PROGRAM AxisDriver
VAR
    fbReset : MC_Reset;  // PLCopen reset
    fbPower : MC_Power;  // PLCopen enable power
    bEnable : BOOL := TRUE;
END_VAR

// Reset faults
fbReset(
    Axis := gVar.gAxis1,
    Execute := bEnable
);

// Enable drive
fbPower(
    Axis := gVar.gAxis1,
    Enable := bEnable,
    Enable_Positive := TRUE,
    Enable_Negative := TRUE
);

END_PROGRAM

(* stored: Version 1.1.0.1
   POU AxisDriver: Id {f302b0f2-58bd-44a5-8d1d-ac1788493a50}, SpecialFunc None *)
